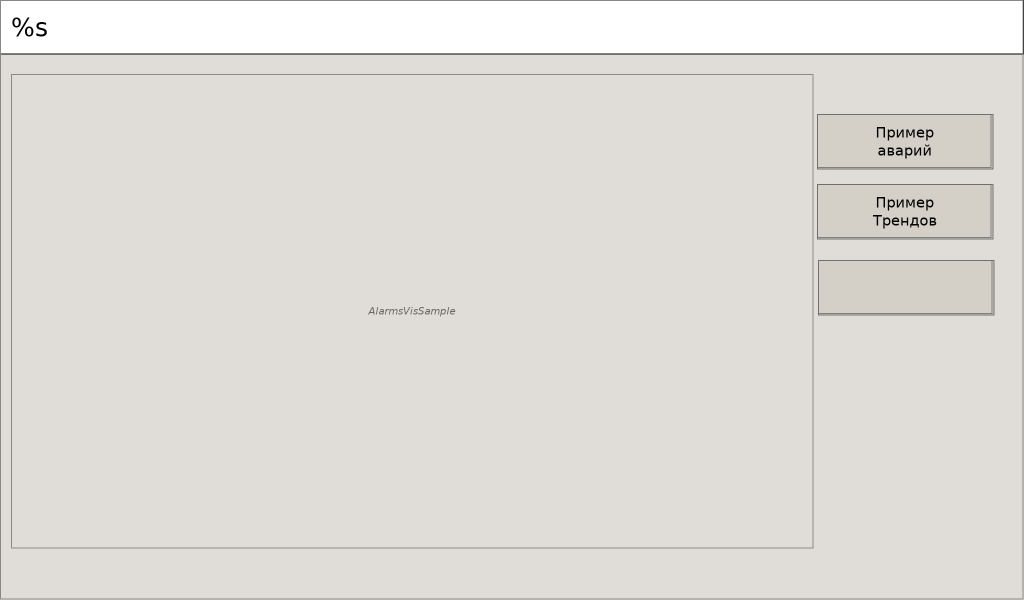
VISUALIZATION Visualization  // 1024x600
    Rectangle (0,0 1024x54), "%s", text variable: Tc3_BAR_Common.LibAlarm.Global_TimeStr
    Frame (11,74 802x474)
        shows AlarmsVisSample()
        shows TrendsSampleVis()
        shows vBrowser()
    Button (817,114 176x55), "Пример аварий"
        OnMouseClick: FrameSelectionChange Selection=SelectedFrame=b3597301-8c91-4ed9-9bbf-06002503f2d3, GlobSel=AssignType=Directly, SelType=Locally
    Button (817,184 176x55), "Пример Трендов"
        OnMouseClick: FrameSelectionChange Selection=SelectedFrame=b3597301-8c91-4ed9-9bbf-06002503f2d3, Selection=1, GlobSel=AssignType=Directly, SelType=Locally
    Button (818,260 176x55)
        OnMouseClick: FrameSelectionChange Selection=SelectedFrame=b3597301-8c91-4ed9-9bbf-06002503f2d3, Selection=2, GlobSel=AssignType=Directly, SelType=Locally
END_VISUALIZATION

(* stored: Version 1.1.0.1, ProductVersion 3.1.4024.10
   Visu Visualization: Id {c30fdee0-db42-47af-85f2-82c391702b8f} *)
